% RSLogix 500 project 1_MOTOR_START_STOP_CONTROL.RSS, saved by version 8.30.00.16 %
PROJECT "PROG_1"    % processor: MicroLogix 1000 %

PROGRAM FILES
  LAD 2   2 rungs
  LAD 3, 4, 5, 6, 7, 8, 9, 10, 11, 12, 13, 14, 15, 16: only END

DATA FILES
  O0 OUTPUT  1 elements
  I1 INPUT  2 elements
  S2 STATUS  33 elements
  B3 BINARY  32 elements
  T4 TIMER  40 elements
  C5 COUNTER  32 elements
  R6 CONTROL  16 elements
  N7 INTEGER  105 elements

LADDER 2
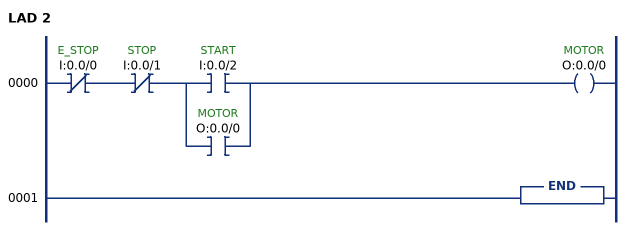
% Rung: 0 %
SOR XIO I:0.0/0 XIO I:0.0/1 BST XIC I:0.0/2 NXB XIC O:0.0/0 BND OTE O:0.0/0 EOR
%   I:0.0/0  E_STOP %
%   I:0.0/1  STOP %
%   I:0.0/2  START %
%   O:0.0/0  MOTOR %
% Rung: 1 %
SOR END EOR

OTHER DOCUMENTED ADDRESSES
  I:0.0/3  J
  O:0.0/1  H
